{attribute addProperty BoxType "EL9560-0000-0016"}
{attribute addProperty Id "Status_UsAT %I*Status_Us_324A4102810Status_UoAT %I*Status_Uo_324A4102810WcStateAT %I*WcState_F855686C1620InfoDataAT %I*InfoData_192954DE1620"}
{attribute addProperty CRC "2031364763"}
{attribute addProperty SizeInBites "48"}
{attribute addProperty SizeInBytes "6"}
TYPE EL9560_A2048F02 :
STRUCT
	{attribute addProperty Name "Status_Us"}
	Status_Us : Status_Us_324A4102;
	{attribute addProperty Name "Status_Uo"}
	Status_Uo : Status_Uo_324A4102;
	{attribute addProperty Name "WcState"}
	WcState : WcState_F855686C;
	{attribute addProperty Name "InfoData"}
	InfoData : InfoData_192954DE;
END_STRUCT
END_TYPE

(* stored: Version 1.2.0.0, ProductVersion 3.1.4024.9
   DUT EL9560_A2048F02: Id {b1c6b60b-40a4-4e22-b5cc-63ba133638ba} *)
